(* IEC 61131-3 sources: st-fmt/tests/fixtures/config, 2 files *)

(* ---- configuration.expected.st ---- *)
CONFIGURATION Plant
VAR_GLOBAL
    gCounter : INT;
END_VAR
RESOURCE Station1 ON CPU001
VAR_GLOBAL
    gLocal : BOOL;
END_VAR
TASK Fast(interval := T#10ms, priority := 1);
TASK Slow(interval := T#1s, priority := 5);
PROGRAM Main WITH Fast : MainProg;
PROGRAM Aux WITH Slow : AuxProg(nInput := 1, bFlag => bResult);
END_RESOURCE
END_CONFIGURATION

(* ---- configuration.st ---- *)
configuration Plant
VAR_GLOBAL
gCounter : INT;
END_VAR
resource Station1 on CPU001
VAR_GLOBAL
gLocal : BOOL;
END_VAR
task Fast(interval := t#10ms, priority := 1);
task Slow(interval := T#1S, priority:=5);
program Main with Fast : MainProg;
program Aux with Slow : AuxProg(nInput := 1, bFlag => bResult);
end_resource
end_configuration
